// TwinCAT 3 PLC project LiquidJetPLC
// ProgramVersion: 3.1.4023.0
// libraries:
//   LCLS General, * (SLAC)
//   lcls-twincat-motion, * (SLAC)
//   PMPS, * (SLAC - LCLS)
//   Tc2_EtherCAT, * (Beckhoff Automation GmbH)
//   Tc2_Standard, * (Beckhoff Automation GmbH)
//   Tc2_System, * (Beckhoff Automation GmbH)
//   Tc3_Module, * (Beckhoff Automation GmbH)
// project tree:
//   / PlcTask.TcTTO
//   POUs/ Main.TcPOU
// real-time tasks:
//   TASK PlcTask: cycle T#10ms, priority 20, ADS port 350
// motion (NC):
//   TASK NC-Task 1 SAF: cycle T#2ms, priority 4, ADS port 501
//   TASK NC-Task 1 SVB: cycle T#10ms, priority 8, ADS port 511
//   AXIS SS_TOP_X_MOT (id 1)
//     Dynamic: AccelerationMaximum=50, DecelerationMaximum=50, Acceleration=23.8095, Deceleration=23.8095, Jerk=70.8615
//     Velo: RefSearch=0.5, RefSync=0.5, SlowManual=0.2, FastManual=0.5, Maximum=1
//     OtherSettings: AllowMotionCmdToSlave=true, PulseDistancePos=0.5, PulseDistanceNeg=0.5
//     encoder EncType=4
//       EncPara: ScaleFactorNumerator=7.8125e-05, Inverse=true, MaxCount=#x0000ffff
//         Inc: RefSoftSyncMask=#x0000ffff
//     drive DrvType=24
//       DrvPara: Inverse=true
//         Analog: VeloReferenz=10, ScaleFactorActTorque=0.1
//         TimeComp: TaskDelayCycles=1
//     controller CtrType=1
//       CtrPara: PriorControlFactor=1
//         PosDiffControl: Range=1
//         Observer: BandWidth=20
//   AXIS SS_TOP_Y_MOT (id 2)
//     Dynamic: AccelerationMaximum=10, DecelerationMaximum=10, Acceleration=5.98802, Deceleration=5.98802, Jerk=17.9282
//     Velo: RefSearch=0.2, RefSync=0.2, SlowManual=0.2, FastManual=0.5, Maximum=0.5
//     OtherSettings: AllowMotionCmdToSlave=true, PulseDistancePos=0.5, PulseDistanceNeg=0.5
//     encoder EncType=4
//       EncPara: ScaleFactorNumerator=1.953125e-05, Inverse=true, MaxCount=#x0000ffff
//         Inc: RefSoftSyncMask=#x0000ffff
//     drive DrvType=24
//       DrvPara: Inverse=true
//         Analog: VeloReferenz=2.5, ScaleFactorActTorque=0.1
//         TimeComp: TaskDelayCycles=1
//     controller CtrType=1
//       CtrPara: PriorControlFactor=1
//         PosDiffControl: Range=0.5
//         Observer: BandWidth=20
//   AXIS SS_BOT_X_MOT (id 3)
//   AXIS SS_BOT_Y_MOT (id 4)
//   AXIS JET_X_MOT (id 5)
//   AXIS JET_Y_MOT (id 6)
//   AXIS JET_Z_MOT (id 7)
//     Dynamic: AccelerationMaximum=50, DecelerationMaximum=50, Acceleration=23.8094883787375, Deceleration=23.8094883787375, Jerk=70.8614671071547
//     Velo: RefSearch=0.5, RefSync=0.5, SlowManual=0.2, FastManual=0.5, Maximum=1
//     OtherSettings: AllowMotionCmdToSlave=true, PulseDistancePos=0.5, PulseDistanceNeg=0.5
//     encoder EncType=4
//       EncPara: MaxCount=#x0000ffff
//         Inc: RefSoftSyncMask=#x0000ffff
//     drive DrvType=24
//       DrvPara: Inverse=true
//         Analog: VeloReferenz=10, ScaleFactorActTorque=0.1
//         TimeComp: TaskDelayCycles=1
//     controller CtrType=1
//       CtrPara: PriorControlFactor=1
//         PosDiffControl: Range=1
//         Observer: BandWidth=20
//   AXIS VH_EPIX_X_MOT (id 8)
//     Dynamic: AccelerationMaximum=50, DecelerationMaximum=50, Acceleration=23.8095, Deceleration=23.8095, Jerk=70.8615
//     Velo: RefSearch=0.1, RefSync=0.1, SlowManual=0.1, FastManual=0.2, Maximum=2
//     OtherSettings: AllowMotionCmdToSlave=true, PulseDistancePos=0.5, PulseDistanceNeg=0.5
//     encoder EncType=4
//       EncPara: ScaleFactorNumerator=0.0002, Inverse=true, MaxCount=#x0000ffff
//         Inc: RefSoftSyncMask=#x0000ffff
//     drive DrvType=24
//       DrvPara: Inverse=true
//         Analog: VeloReferenz=10, ScaleFactorActTorque=0.1
//         TimeComp: TaskDelayCycles=1
//     controller CtrType=1
//       CtrPara: PriorControlFactor=1
//         PosDiffControl: Range=0.5
//         Observer: BandWidth=20
// I/O:
//   DEVICE Device 1 (EtherCAT)
// variable links:
//   (this object) <-> Device 1 (EtherCAT)/E0 (EK1200)/E7 (EK1122)/E20 (EK1100)/E21 (EL7041)
//     Drive/Inputs/In/nState1 @bit 3 <-> STM Status/Status/Error
//     Drive/Inputs/In/nState1 @bit 5 <-> STM Status/Status/Moving negative
//     Drive/Inputs/In/nState1 @bit 4 <-> STM Status/Status/Moving positive
//     Drive/Inputs/In/nState1 @bit 1 <-> STM Status/Status/Ready
//     Drive/Inputs/In/nState1 <-> STM Status/Status/Ready to enable
//     Drive/Inputs/In/nState1 @bit 6 <-> STM Status/Status/Torque reduced
//     Drive/Inputs/In/nState1 @bit 2 <-> STM Status/Status/Warning
//     Drive/Inputs/In/nState2 @bit 3 <-> STM Status/Status/Digital input 1
//     Drive/Inputs/In/nState2 @bit 4 <-> STM Status/Status/Digital input 2
//     Drive/Inputs/In/nState2 @bit 5 <-> STM Status/Status/Sync error
//     Drive/Inputs/In/nState2 @bit 7 <-> STM Status/Status/TxPDO Toggle
//     Drive/Inputs/In/nState4 @bit 1 <-> WcState/InputToggle
//     Drive/Inputs/In/nState4 <-> WcState/WcState
//     Drive/Outputs/Out/nCtrl1 <-> STM Control/Control/Enable
//     Drive/Outputs/Out/nCtrl1 @bit 2 <-> STM Control/Control/Reduce torque
//     Drive/Outputs/Out/nCtrl1 @bit 1 <-> STM Control/Control/Reset
//     Drive/Outputs/Out/nDataOut2[0] <-> STM Velocity/Velocity
//     Enc/Inputs/In/nDataIn1[0] <-> ENC Status compact/Counter value
//     Enc/Inputs/In/nDataIn2[0] <-> ENC Status compact/Latch value
//     Enc/Inputs/In/nState1 @bit 4 <-> ENC Status compact/Status/Counter overflow
//     Enc/Inputs/In/nState1 @bit 3 <-> ENC Status compact/Status/Counter underflow
//     Enc/Inputs/In/nState1 @bit 7 <-> ENC Status compact/Status/Extrapolation stall
//     Enc/Inputs/In/nState1 <-> ENC Status compact/Status/Latch C valid
//     Enc/Inputs/In/nState1 @bit 1 <-> ENC Status compact/Status/Latch extern valid
//     Enc/Inputs/In/nState1 @bit 2 <-> ENC Status compact/Status/Set counter done
//     Enc/Inputs/In/nState2 @bit 4 <-> ENC Status compact/Status/Status of extern latch
//     Enc/Inputs/In/nState2 <-> ENC Status compact/Status/Status of input A
//     Enc/Inputs/In/nState2 @bit 1 <-> ENC Status compact/Status/Status of input B
//     Enc/Inputs/In/nState2 @bit 2 <-> ENC Status compact/Status/Status of input C
//     Enc/Inputs/In/nState2 @bit 5 <-> ENC Status compact/Status/Sync error
//     Enc/Inputs/In/nState2 @bit 7 <-> ENC Status compact/Status/TxPDO Toggle
//     Enc/Inputs/In/nState4 @bit 1 <-> WcState/InputToggle
//     Enc/Inputs/In/nState4 <-> WcState/WcState
//     Enc/Outputs/Out/nCtrl1 <-> ENC Control compact/Control/Enable latch C
//     Enc/Outputs/Out/nCtrl1 @bit 3 <-> ENC Control compact/Control/Enable latch extern on negative edge
//     Enc/Outputs/Out/nCtrl1 @bit 1 <-> ENC Control compact/Control/Enable latch extern on positive edge
//     Enc/Outputs/Out/nCtrl1 @bit 2 <-> ENC Control compact/Control/Set counter
//     Enc/Outputs/Out/nDataOut1[0] <-> ENC Control compact/Set counter value
//   (this object) <-> Device 1 (EtherCAT)/E0 (EK1200)/E7 (EK1122)/E20 (EK1100)/E23 (EL7041)
//     Drive/Inputs/In/nState1 @bit 3 <-> STM Status/Status/Error
//     Drive/Inputs/In/nState1 @bit 5 <-> STM Status/Status/Moving negative
//     Drive/Inputs/In/nState1 @bit 4 <-> STM Status/Status/Moving positive
//     Drive/Inputs/In/nState1 @bit 1 <-> STM Status/Status/Ready
//     Drive/Inputs/In/nState1 <-> STM Status/Status/Ready to enable
//     Drive/Inputs/In/nState1 @bit 6 <-> STM Status/Status/Torque reduced
//     Drive/Inputs/In/nState1 @bit 2 <-> STM Status/Status/Warning
//     Drive/Inputs/In/nState2 @bit 3 <-> STM Status/Status/Digital input 1
//     Drive/Inputs/In/nState2 @bit 4 <-> STM Status/Status/Digital input 2
//     Drive/Inputs/In/nState2 @bit 5 <-> STM Status/Status/Sync error
//     Drive/Inputs/In/nState2 @bit 7 <-> STM Status/Status/TxPDO Toggle
//     Drive/Inputs/In/nState4 @bit 1 <-> WcState/InputToggle
//     Drive/Inputs/In/nState4 <-> WcState/WcState
//     Drive/Outputs/Out/nCtrl1 <-> STM Control/Control/Enable
//     Drive/Outputs/Out/nCtrl1 @bit 2 <-> STM Control/Control/Reduce torque
//     Drive/Outputs/Out/nCtrl1 @bit 1 <-> STM Control/Control/Reset
//     Drive/Outputs/Out/nDataOut2[0] <-> STM Velocity/Velocity
//     Enc/Inputs/In/nDataIn1[0] <-> ENC Status compact/Counter value
//     Enc/Inputs/In/nDataIn2[0] <-> ENC Status compact/Latch value
//     Enc/Inputs/In/nState1 @bit 4 <-> ENC Status compact/Status/Counter overflow
//     Enc/Inputs/In/nState1 @bit 3 <-> ENC Status compact/Status/Counter underflow
//     Enc/Inputs/In/nState1 @bit 7 <-> ENC Status compact/Status/Extrapolation stall
//     Enc/Inputs/In/nState1 <-> ENC Status compact/Status/Latch C valid
//     Enc/Inputs/In/nState1 @bit 1 <-> ENC Status compact/Status/Latch extern valid
//     Enc/Inputs/In/nState1 @bit 2 <-> ENC Status compact/Status/Set counter done
//     Enc/Inputs/In/nState2 @bit 4 <-> ENC Status compact/Status/Status of extern latch
//     Enc/Inputs/In/nState2 <-> ENC Status compact/Status/Status of input A
//     Enc/Inputs/In/nState2 @bit 1 <-> ENC Status compact/Status/Status of input B
//     Enc/Inputs/In/nState2 @bit 2 <-> ENC Status compact/Status/Status of input C
//     Enc/Inputs/In/nState2 @bit 5 <-> ENC Status compact/Status/Sync error
//     Enc/Inputs/In/nState2 @bit 7 <-> ENC Status compact/Status/TxPDO Toggle
//     Enc/Inputs/In/nState4 @bit 1 <-> WcState/InputToggle
//     Enc/Inputs/In/nState4 <-> WcState/WcState
//     Enc/Outputs/Out/nCtrl1 <-> ENC Control compact/Control/Enable latch C
//     Enc/Outputs/Out/nCtrl1 @bit 3 <-> ENC Control compact/Control/Enable latch extern on negative edge
//     Enc/Outputs/Out/nCtrl1 @bit 1 <-> ENC Control compact/Control/Enable latch extern on positive edge
//     Enc/Outputs/Out/nCtrl1 @bit 2 <-> ENC Control compact/Control/Set counter
//     Enc/Outputs/Out/nDataOut1[0] <-> ENC Control compact/Set counter value
//   (this object) <-> Device 1 (EtherCAT)/E0 (EK1200)/E3 (EL5101)
//     Enc/Inputs/In/nDataIn1[0] <-> ENC Status compact/Counter value
//     Enc/Inputs/In/nDataIn2[0] <-> ENC Status compact/Latch value
//     Enc/Inputs/In/nState1 @bit 4 <-> ENC Status compact/Status/Counter overflow
//     Enc/Inputs/In/nState1 @bit 3 <-> ENC Status compact/Status/Counter underflow
//     Enc/Inputs/In/nState1 @bit 7 <-> ENC Status compact/Status/Extrapolation stall
//     Enc/Inputs/In/nState1 <-> ENC Status compact/Status/Latch C valid
//     Enc/Inputs/In/nState1 @bit 1 <-> ENC Status compact/Status/Latch extern valid
//     Enc/Inputs/In/nState1 @bit 6 <-> ENC Status compact/Status/Open circuit
//     Enc/Inputs/In/nState1 @bit 2 <-> ENC Status compact/Status/Set counter done
//     Enc/Inputs/In/nState1 @bit 5 <-> ENC Status compact/Status/Status of input status
//     Enc/Inputs/In/nState2 @bit 4 <-> ENC Status compact/Status/Status of extern latch
//     Enc/Inputs/In/nState2 <-> ENC Status compact/Status/Status of input A
//     Enc/Inputs/In/nState2 @bit 1 <-> ENC Status compact/Status/Status of input B
//     Enc/Inputs/In/nState2 @bit 2 <-> ENC Status compact/Status/Status of input C
//     Enc/Inputs/In/nState2 @bit 3 <-> ENC Status compact/Status/Status of input gate
//     Enc/Inputs/In/nState2 @bit 5 <-> ENC Status compact/Status/Sync error
//     Enc/Inputs/In/nState2 @bit 6 <-> ENC Status compact/Status/TxPDO State
//     Enc/Inputs/In/nState2 @bit 7 <-> ENC Status compact/Status/TxPDO Toggle
//     Enc/Inputs/In/nState4 @bit 1 <-> WcState/InputToggle
//     Enc/Inputs/In/nState4 <-> WcState/WcState
//     Enc/Outputs/Out/nCtrl1 <-> ENC Control compact/Control/Enable latch C
//     Enc/Outputs/Out/nCtrl1 @bit 3 <-> ENC Control compact/Control/Enable latch extern on negative edge
//     Enc/Outputs/Out/nCtrl1 @bit 1 <-> ENC Control compact/Control/Enable latch extern on positive edge
//     Enc/Outputs/Out/nCtrl1 @bit 2 <-> ENC Control compact/Control/Set counter
//     Enc/Outputs/Out/nDataOut1[0] <-> ENC Control compact/Set counter value
//   (this object) <-> Device 1 (EtherCAT)/E0 (EK1200)/E7 (EK1122)/E20 (EK1100)/E30 (EL7041)
//     Drive/Inputs/In/nState1 @bit 3 <-> STM Status/Status/Error
//     Drive/Inputs/In/nState1 @bit 5 <-> STM Status/Status/Moving negative
//     Drive/Inputs/In/nState1 @bit 4 <-> STM Status/Status/Moving positive
//     Drive/Inputs/In/nState1 @bit 1 <-> STM Status/Status/Ready
//     Drive/Inputs/In/nState1 <-> STM Status/Status/Ready to enable
//     Drive/Inputs/In/nState1 @bit 6 <-> STM Status/Status/Torque reduced
//     Drive/Inputs/In/nState1 @bit 2 <-> STM Status/Status/Warning
//     Drive/Inputs/In/nState2 @bit 3 <-> STM Status/Status/Digital input 1
//     Drive/Inputs/In/nState2 @bit 4 <-> STM Status/Status/Digital input 2
//     Drive/Inputs/In/nState2 @bit 5 <-> STM Status/Status/Sync error
//     Drive/Inputs/In/nState2 @bit 7 <-> STM Status/Status/TxPDO Toggle
//     Drive/Inputs/In/nState4 @bit 1 <-> WcState/InputToggle
//     Drive/Inputs/In/nState4 <-> WcState/WcState
//     Drive/Outputs/Out/nCtrl1 <-> STM Control/Control/Enable
//     Drive/Outputs/Out/nCtrl1 @bit 2 <-> STM Control/Control/Reduce torque
//     Drive/Outputs/Out/nCtrl1 @bit 1 <-> STM Control/Control/Reset
//     Drive/Outputs/Out/nDataOut2[0] <-> STM Velocity/Velocity
//   (this object) <-> Device 1 (EtherCAT)/E0 (EK1200)/E4 (EL5101)
//     Enc/Inputs/In/nDataIn1[0] <-> ENC Status compact/Counter value
//     Enc/Inputs/In/nDataIn2[0] <-> ENC Status compact/Latch value
//     Enc/Inputs/In/nState1 @bit 4 <-> ENC Status compact/Status/Counter overflow
//     Enc/Inputs/In/nState1 @bit 3 <-> ENC Status compact/Status/Counter underflow
//     Enc/Inputs/In/nState1 @bit 7 <-> ENC Status compact/Status/Extrapolation stall
//     Enc/Inputs/In/nState1 <-> ENC Status compact/Status/Latch C valid
//     Enc/Inputs/In/nState1 @bit 1 <-> ENC Status compact/Status/Latch extern valid
//     Enc/Inputs/In/nState1 @bit 6 <-> ENC Status compact/Status/Open circuit
//     Enc/Inputs/In/nState1 @bit 2 <-> ENC Status compact/Status/Set counter done
//     Enc/Inputs/In/nState1 @bit 5 <-> ENC Status compact/Status/Status of input status
//     Enc/Inputs/In/nState2 @bit 4 <-> ENC Status compact/Status/Status of extern latch
//     Enc/Inputs/In/nState2 <-> ENC Status compact/Status/Status of input A
//     Enc/Inputs/In/nState2 @bit 1 <-> ENC Status compact/Status/Status of input B
//     Enc/Inputs/In/nState2 @bit 2 <-> ENC Status compact/Status/Status of input C
//     Enc/Inputs/In/nState2 @bit 3 <-> ENC Status compact/Status/Status of input gate
//     Enc/Inputs/In/nState2 @bit 5 <-> ENC Status compact/Status/Sync error
//     Enc/Inputs/In/nState2 @bit 6 <-> ENC Status compact/Status/TxPDO State
//     Enc/Inputs/In/nState2 @bit 7 <-> ENC Status compact/Status/TxPDO Toggle
//     Enc/Inputs/In/nState4 @bit 1 <-> WcState/InputToggle
//     Enc/Inputs/In/nState4 <-> WcState/WcState
//     Enc/Outputs/Out/nCtrl1 <-> ENC Control compact/Control/Enable latch C
//     Enc/Outputs/Out/nCtrl1 @bit 3 <-> ENC Control compact/Control/Enable latch extern on negative edge
//     Enc/Outputs/Out/nCtrl1 @bit 1 <-> ENC Control compact/Control/Enable latch extern on positive edge
//     Enc/Outputs/Out/nCtrl1 @bit 2 <-> ENC Control compact/Control/Set counter
//     Enc/Outputs/Out/nDataOut1[0] <-> ENC Control compact/Set counter value
//   (this object) <-> Device 1 (EtherCAT)/E0 (EK1200)/E7 (EK1122)/E20 (EK1100)/E31 (EL7041)
//     Drive/Inputs/In/nState1 @bit 3 <-> STM Status/Status/Error
//     Drive/Inputs/In/nState1 @bit 5 <-> STM Status/Status/Moving negative
//     Drive/Inputs/In/nState1 @bit 4 <-> STM Status/Status/Moving positive
//     Drive/Inputs/In/nState1 @bit 1 <-> STM Status/Status/Ready
//     Drive/Inputs/In/nState1 <-> STM Status/Status/Ready to enable
//     Drive/Inputs/In/nState1 @bit 6 <-> STM Status/Status/Torque reduced
//     Drive/Inputs/In/nState1 @bit 2 <-> STM Status/Status/Warning
//     Drive/Inputs/In/nState2 @bit 3 <-> STM Status/Status/Digital input 1
//     Drive/Inputs/In/nState2 @bit 4 <-> STM Status/Status/Digital input 2
//     Drive/Inputs/In/nState2 @bit 5 <-> STM Status/Status/Sync error
//     Drive/Inputs/In/nState2 @bit 7 <-> STM Status/Status/TxPDO Toggle
//     Drive/Inputs/In/nState4 @bit 1 <-> WcState/InputToggle
//     Drive/Inputs/In/nState4 <-> WcState/WcState
//     Drive/Outputs/Out/nCtrl1 <-> STM Control/Control/Enable
//     Drive/Outputs/Out/nCtrl1 @bit 2 <-> STM Control/Control/Reduce torque
//     Drive/Outputs/Out/nCtrl1 @bit 1 <-> STM Control/Control/Reset
//     Drive/Outputs/Out/nDataOut2[0] <-> STM Velocity/Velocity
//   LiquidJetPLC Instance <-> Device 1 (EtherCAT)/E0 (EK1200)/E5 (EL2004)
//     PlcTask Outputs/Main.bGigePower <-> Channel 1/Output
//   LiquidJetPLC Instance <-> Device 1 (EtherCAT)/E0 (EK1200)/E7 (EK1122)/E20 (EK1100)/E22 (EL1088)
//     PlcTask Inputs/Main.M1.bHome <-> Channel 5/Input
//     PlcTask Inputs/Main.M2.bHome <-> Channel 6/Input
//     PlcTask Inputs/Main.M1.bLimitBackwardEnable <-> Channel 3/Input
//     PlcTask Inputs/Main.M2.bLimitBackwardEnable <-> Channel 4/Input
//     PlcTask Inputs/Main.M1.bLimitForwardEnable <-> Channel 1/Input
//     PlcTask Inputs/Main.M2.bLimitForwardEnable <-> Channel 2/Input
//   LiquidJetPLC Instance <-> Device 1 (EtherCAT)/E0 (EK1200)/E7 (EK1122)/E20 (EK1100)/E25 (EL1088)
//     PlcTask Inputs/Main.M3.bHome <-> Channel 5/Input
//     PlcTask Inputs/Main.M4.bHome <-> Channel 6/Input
//     PlcTask Inputs/Main.M3.bLimitBackwardEnable <-> Channel 3/Input
//     PlcTask Inputs/Main.M4.bLimitBackwardEnable <-> Channel 4/Input
//     PlcTask Inputs/Main.M3.bLimitForwardEnable <-> Channel 1/Input
//     PlcTask Inputs/Main.M4.bLimitForwardEnable <-> Channel 2/Input
//   LiquidJetPLC Instance <-> Device 1 (EtherCAT)/E0 (EK1200)/E7 (EK1122)/E20 (EK1100)/E29 (EL1088)
//     PlcTask Inputs/Main.M5.bLimitBackwardEnable <-> Channel 1/Input
//     PlcTask Inputs/Main.M6.bLimitBackwardEnable <-> Channel 7/Input
//     PlcTask Inputs/Main.M7.bLimitBackwardEnable <-> Channel 4/Input
//     PlcTask Inputs/Main.M8.bLimitBackwardEnable <-> Channel 6/Input
//     PlcTask Inputs/Main.M5.bLimitForwardEnable <-> Channel 3/Input
//     PlcTask Inputs/Main.M6.bLimitForwardEnable <-> Channel 5/Input
//     PlcTask Inputs/Main.M7.bLimitForwardEnable <-> Channel 2/Input
//     PlcTask Inputs/Main.M8.bLimitForwardEnable <-> Channel 8/Input
//   LiquidJetPLC Instance <-> NC-Task 1 SAF/Axes/JET_X_MOT
//     PlcTask Inputs/Main.M5.Axis.NcToPlc <-> Outputs/ToPlc
//     PlcTask Outputs/Main.M5.Axis.PlcToNc <-> Inputs/FromPlc
//   LiquidJetPLC Instance <-> NC-Task 1 SAF/Axes/JET_Y_MOT
//     PlcTask Inputs/Main.M6.Axis.NcToPlc <-> Outputs/ToPlc
//     PlcTask Outputs/Main.M6.Axis.PlcToNc <-> Inputs/FromPlc
//   LiquidJetPLC Instance <-> NC-Task 1 SAF/Axes/JET_Z_MOT
//     PlcTask Inputs/Main.M7.Axis.NcToPlc <-> Outputs/ToPlc
//     PlcTask Outputs/Main.M7.Axis.PlcToNc <-> Inputs/FromPlc
//   LiquidJetPLC Instance <-> NC-Task 1 SAF/Axes/SS_BOT_X_MOT
//     PlcTask Inputs/Main.M3.Axis.NcToPlc <-> Outputs/ToPlc
//     PlcTask Outputs/Main.M3.Axis.PlcToNc <-> Inputs/FromPlc
//   LiquidJetPLC Instance <-> NC-Task 1 SAF/Axes/SS_BOT_Y_MOT
//     PlcTask Inputs/Main.M4.Axis.NcToPlc <-> Outputs/ToPlc
//     PlcTask Outputs/Main.M4.Axis.PlcToNc <-> Inputs/FromPlc
//   LiquidJetPLC Instance <-> NC-Task 1 SAF/Axes/SS_TOP_X_MOT
//     PlcTask Inputs/Main.M1.Axis.NcToPlc <-> Outputs/ToPlc
//     PlcTask Outputs/Main.M1.Axis.PlcToNc <-> Inputs/FromPlc
//   LiquidJetPLC Instance <-> NC-Task 1 SAF/Axes/SS_TOP_Y_MOT
//     PlcTask Inputs/Main.M2.Axis.NcToPlc <-> Outputs/ToPlc
//     PlcTask Outputs/Main.M2.Axis.PlcToNc <-> Inputs/FromPlc
//   LiquidJetPLC Instance <-> NC-Task 1 SAF/Axes/VH_EPIX_X_MOT
//     PlcTask Inputs/Main.M8.Axis.NcToPlc <-> Outputs/ToPlc
//     PlcTask Outputs/Main.M8.Axis.PlcToNc <-> Inputs/FromPlc

CONFIGURATION LiquidJetPLC
    RESOURCE PLC ON TwinCAT3
        TASK PlcTask(INTERVAL := T#10ms, PRIORITY := 20);
        PROGRAM Main WITH PlcTask : Main;
    END_RESOURCE
END_CONFIGURATION

// ---- POUs/Main.TcPOU
PROGRAM Main
VAR
    {attribute 'pytmc' := 'pv: XCS:LJH:SS:TOP_X'}
    {attribute 'TcLinkTo' := '
        .bLimitForwardEnable	:= TIIB[EL1088_01_22]^Channel 1^Input;
        .bLimitBackwardEnable	:= TIIB[EL1088_01_22]^Channel 3^Input;
        .bHome					:= TIIB[EL1088_01_22]^Channel 5^Input'}
    M1	: ST_MotionStage:= (sName := 'XCS:LJH:SS:TOP_X'); //SS_TOP_X_MOT

    {attribute 'pytmc' := 'pv: XCS:LJH:SS:TOP_Y'}
    {attribute 'TcLinkTo' := '
        .bLimitForwardEnable	:= TIIB[EL1088_01_22]^Channel 2^Input;
        .bLimitBackwardEnable	:= TIIB[EL1088_01_22]^Channel 4^Input;
        .bHome					:= TIIB[EL1088_01_22]^Channel 6^Input'}
    M2	: ST_MotionStage:= (sName := 'XCS:LJH:SS:TOP_Y'); //SS_TOP_Y_MOT

    {attribute 'pytmc' := 'pv: XCS:LJH:SS:BOT_X'}
    {attribute 'TcLinkTo' := '
        .bLimitForwardEnable	:= TIIB[EL1088_01_25]^Channel 1^Input;
        .bLimitBackwardEnable	:= TIIB[EL1088_01_25]^Channel 3^Input;
        .bHome					:= TIIB[EL1088_01_25]^Channel 5^Input'}
    M3	: ST_MotionStage:= (sName := 'XCS:LJH:SS:BOT_X'); //SS_BOT_X_MOT

    {attribute 'pytmc' := 'pv: XCS:LJH:SS:BOT_Y'}
    {attribute 'TcLinkTo' := '
        .bLimitForwardEnable	:= TIIB[EL1088_01_25]^Channel 2^Input;
        .bLimitBackwardEnable	:= TIIB[EL1088_01_25]^Channel 4^Input;
        .bHome					:= TIIB[EL1088_01_25]^Channel 6^Input'}
    M4	: ST_MotionStage:= (sName := 'XCS:LJH:SS:BOT_Y'); //SS_BOT_Y_MOT

    {attribute 'pytmc' := 'pv: XCS:LJH:JET:X'}
    {attribute 'TcLinkTo' := '
        .bLimitBackwardEnable	:= TIIB[EL1088_01_29]^Channel 1^Input;
        .bLimitForwardEnable	:= TIIB[EL1088_01_29]^Channel 3^Input'}
    M5	: ST_MotionStage:= (sName := 'XCS:LJH:JET:X'); //JET_X_MOT

    {attribute 'pytmc' := 'pv: XCS:LJH:JET:Y'}
    {attribute 'TcLinkTo' := '
        .bLimitForwardEnable	:= TIIB[EL1088_01_29]^Channel 5^Input;
        .bLimitBackwardEnable	:= TIIB[EL1088_01_29]^Channel 7^Input'}
    M6	: ST_MotionStage:= (sName := 'XCS:LJH:JET:Y'); //JET_Y_MOT

    {attribute 'pytmc' := 'pv: XCS:LJH:JET:Z'}
    {attribute 'TcLinkTo' := '
        .bLimitForwardEnable	:= TIIB[EL1088_01_29]^Channel 2^Input;
        .bLimitBackwardEnable	:= TIIB[EL1088_01_29]^Channel 4^Input'}
    M7	: ST_MotionStage:= (sName := 'XCS:LJH:JET:Z'); //JET_Z_MOT

    {attribute 'pytmc' := 'pv: XCS:LJH:DET:X'}
    {attribute 'TcLinkTo' := '
        .bLimitBackwardEnable	:= TIIB[EL1088_01_29]^Channel 6^Input;
        .bLimitForwardEnable	:= TIIB[EL1088_01_29]^Channel 8^Input'}
    M8: ST_MotionStage:= (sName := 'XCS:LJH:DET:X') ; //VH_EPIX_X_MOT

    fb_SS_TOP_X	: FB_MotionStage;
    fb_SS_TOP_Y	: FB_MotionStage;
    fb_SS_BOT_X	: FB_MotionStage;
    fb_SS_BOT_Y	: FB_MotionStage;
    fb_JET_X	: FB_MotionStage;
    fb_JET_Y	: FB_MotionStage;
    fb_JET_Z	: FB_MotionStage;
    fb_VH_EPIX_X: FB_MotionStage;

    bInit: BOOL := TRUE;

END_VAR


//fbMotion
fb_SS_TOP_X(stMotionStage := M1);
fb_SS_TOP_Y(stMotionStage := M2);
fb_SS_BOT_X(stMotionStage := M3);
fb_SS_BOT_Y(stMotionStage := M4);
fb_JET_X(stMotionStage := M5);
fb_JET_Y(stMotionStage := M6);
fb_JET_Z(stMotionStage := M7);
fb_VH_EPIX_X(stMotionStage := M8);

IF bInit THEN
    bInit := FALSE;

    M1.bHardwareEnable := TRUE;
    M1.bPowerSelf      := TRUE;
    M1.fVelocity       := 0.1;
    M1.nEnableMode     := E_StageEnableMode.DURING_MOTION;
    M1.nBrakeMode      := E_StageBrakeMode.NO_BRAKE;
    M1.nHomingMode     := E_EpicsHomeCmd.LOW_LIMIT;
    M1.fHomePosition   := 0;

    M2.bHardwareEnable := TRUE;
    M2.bPowerSelf      := TRUE;
    M2.fVelocity       := 0.1;
    M2.nEnableMode     := E_StageEnableMode.DURING_MOTION;
    M2.nBrakeMode      := E_StageBrakeMode.NO_BRAKE;
    M2.nHomingMode     := E_EpicsHomeCmd.HIGH_LIMIT;
    M2.fHomePosition   := 5.87;

    M3.bHardwareEnable := TRUE;
    M3.bPowerSelf      := TRUE;
    M3.fVelocity       := 0.1;
    M3.nEnableMode     := E_StageEnableMode.DURING_MOTION;
    M3.nBrakeMode      := E_StageBrakeMode.NO_BRAKE;
    M3.nHomingMode     := E_EpicsHomeCmd.LOW_LIMIT;
    M3.fHomePosition   := 0;

    M4.bHardwareEnable := TRUE;
    M4.bPowerSelf      := TRUE;
    M4.fVelocity       := 0.1;
    M4.nEnableMode     := E_StageEnableMode.DURING_MOTION;
    M4.nBrakeMode      := E_StageBrakeMode.NO_BRAKE;
    M4.nHomingMode     := E_EpicsHomeCmd.HIGH_LIMIT;
    M4.fHomePosition   := 5.25;

    M5.bHardwareEnable := TRUE;
    M5.bPowerSelf      := TRUE;
    M5.fVelocity       := 0.1;
    M5.nEnableMode     := E_StageEnableMode.DURING_MOTION;
    M5.nBrakeMode      := E_StageBrakeMode.NO_BRAKE;
    M5.nHomingMode     := E_EpicsHomeCmd.HIGH_LIMIT;
    M5.fHomePosition   := 0;

    M6.bHardwareEnable := TRUE;
    M6.bPowerSelf      := TRUE;
    M6.fVelocity       := 0.1;
    M6.nEnableMode     := E_StageEnableMode.DURING_MOTION;
    M6.nBrakeMode      := E_StageBrakeMode.NO_BRAKE;
    M6.nHomingMode     := E_EpicsHomeCmd.LOW_LIMIT;
    M6.fHomePosition   := 0;

    M7.bHardwareEnable := TRUE;
    M7.bPowerSelf      := TRUE;
    M7.fVelocity       := 0.1;
    M7.nEnableMode     := E_StageEnableMode.DURING_MOTION;
    M7.nBrakeMode      := E_StageBrakeMode.NO_BRAKE;
    M7.nHomingMode     := E_EpicsHomeCmd.LOW_LIMIT;
    M7.fHomePosition   := 0;

    M8.bHardwareEnable := TRUE;
    M8.bPowerSelf      := TRUE;
    M8.fVelocity       := 0.1;
    M8.nEnableMode     := E_StageEnableMode.DURING_MOTION;
    M8.nBrakeMode      := E_StageBrakeMode.NO_BRAKE;
    M8.nHomingMode     := E_EpicsHomeCmd.LOW_LIMIT;
    M8.fHomePosition   := 0;
END_IF

END_PROGRAM
